FUNCTION F_ComputeRawVarint32Size : UDINT
VAR_INPUT
    nValue : UDINT;
END_VAR
VAR
    i       : UDINT;
END_VAR


FOR i := 1 TO 4 DO    
    IF (nValue AND SHL(16#FFFFFFFF, 7 * i)) = 0 THEN
        F_ComputeRawVarint32Size := i;
        RETURN;
    END_IF
END_FOR

F_ComputeRawVarint32Size := 5;

END_FUNCTION

(* stored: Version 1.1.0.1
   POU F_ComputeRawVarint32Size: Id {57596d0e-64a9-4d90-9368-4e0606fc753f}, SpecialFunc None *)
